PROGRAM MAIN
VAR
END_VAR

Tcp_ip();

END_PROGRAM

(* stored: Version 1.1.0.1, ProductVersion 3.1.4024.0
   POU MAIN: Id {28764a43-5ca1-4b93-894f-ebafd72f86c6}, SpecialFunc None *)
